// TwinCAT 3 PLC project LabExercise
// ProgramVersion: 3.1.4023.0
// libraries:
//   Tc2_NCI, * (Beckhoff Automation GmbH)
//   Tc2_Standard, * (Beckhoff Automation GmbH)
//   Tc2_System, * (Beckhoff Automation GmbH)
//   Tc3_Module, * (Beckhoff Automation GmbH)
//   VisuDialogs, * (System)
// project tree:
//   Comissioning/Function blocks/ FB_ModifyAutomaticControlSettings.TcPOU (not stored)
//   Comissioning/GVLs/ G_Commissioning.TcGVL (not stored)
//   Comissioning/Struct/ ST_AutomaticControlSettings.TcDUT (not stored), ST_ClosedLoopControlSettings.TcDUT (not stored), ST_MotionReferenceGeneratorSettings.TcDUT (not stored), ST_OpenLoopControlSettings.TcDUT (not stored)
//   ControlBox/Interfaces/ I_ControlBox.TcIO (not stored)
//   ControlBox/Function blocks/ FB_ControlBox.TcPOU, FB_RealControlBox.TcPOU (not stored), FB_VirtualControlBox.TcPOU (not stored)
//   CraneControl/Function blocks/Sub blocks/ FB_ActiveDamping.TcPOU (not stored), FB_Clock.TcPOU (not stored), FB_ClosedLoopControl.TcPOU (not stored), FB_Joystick.TcPOU (not stored), FB_MotionReferenceGenerator_limit.TcPOU (not stored), FB_OpenLoopControl.TcPOU (not stored), FB_ResetIntegralController.TcPOU (not stored), FB_Status.TcPOU (not stored)
//   CraneControl/Enums/ E_Mode.TcDUT (not stored), E_Status.TcDUT (not stored)
//   CraneControl/Function blocks/Main blocks/ FB_AutomaticControl.TcPOU (not stored), FB_ManualControl.TcPOU (not stored)
//   CraneControl/Functions/ F_BarToEng.TcPOU (not stored), F_LminToEng.TcPOU (not stored), F_RadToDeg.TcPOU (not stored)
//   CraneControl/GVLs/ G_Parameters.TcGVL (not stored), G_Work.TcGVL (not stored)
//   CraneControl/Struct/ ST_ActiveDamping.TcDUT (not stored), ST_Parameters.TcDUT (not stored)
//   / GlobalTextList.TcGTLO (not stored), PlcTask.TcTTO (not stored), Simulator.TcTTO (not stored), Visualization Manager.TcVMO (not stored)
//   HMI/ HMI.TcVIS (not stored)
//   HMI/Sub/ CommissioningHMI.TcVIS (not stored), VirtualControlBox.TcVIS (not stored)
//   Inputs/ FB_JoystickInputScaling.TcPOU (not stored), FB_PositionInputScaling.TcPOU (not stored), FB_PressureInputScaling.TcPOU (not stored), G_Inputs.TcGVL (not stored), G_Sensors.TcGVL (not stored)
//   Inputs/Struct/ ST_AnalogInput.TcDUT (not stored), ST_AnalogInputStatus.TcDUT (not stored)
//   Internship/ FB_ControlBlock.TcPOU, FB_SpeedProfile.TcPOU, F_PressureSensorInToBar.TcPOU (not stored), GVL_191759331.TcGVL, V2Q2u.TcPOU (not stored)
//   Outputs/ FB_ValveOutput.TcPOU (not stored), G_Outputs.TcGVL (not stored)
//   Outputs/Struct/ ST_pValveDeadBand.TcDUT (not stored), ST_ValveOutput.TcDUT (not stored)
//   ControlBox/GVLs/ G_VirtualControlBox.TcGVL (not stored)
//   Programs/ MAIN.TcPOU (not stored), P_ControlBlock.TcPOU, P_Commissioning.TcPOU (not stored), P_ControlBox.TcPOU (not stored), P_CraneControl.TcPOU (not stored), P_Inputs.TcPOU (not stored), P_OutputNonCompensated.TcPOU (not stored), P_Outputs.TcPOU (not stored), P_Simulator.TcPOU
//   Simulator/ FB_CraneSimulator.TcPOU (not stored), G_Simulator.TcGVL (not stored)
// real-time tasks:
//   TASK PlcTask: cycle T#1ms, priority 20, ADS port 350
//   TASK Simulator: cycle T#100us, priority 1, ADS port 351
// I/O:
//   DEVICE Device 5 (EtherCAT), AmsNetId 10.229.3.117.6.1
//     RIO (EK1100) [EK1100 EtherCAT Coupler (2A E-Bus)]
//       DI (EL1008) [EL1008 8Ch. Dig. Input 24V, 3ms]
//       DO (EL2008) [EL2008 8Ch. Dig. Output 24V, 0.5A]
//       AI1 (EL3068) [EL3068 8Ch. Ana. Input 0-10V]
//       AI2 (EL3068) [EL3068 8Ch. Ana. Input 0-10V]
//       AI3 (EL3174) [EL3174 4Ch. Ana. Input +/-10V Diff., +/-20mA SingleEnded, 16 Bit]
//       AO (EL4104) [EL4104 4Ch. Ana. Output 0-10V, 16bit]
//       End Cap (EL9011) [EL9011 End Terminal]
// variable links:
//   LabExercise/LabExercise Instance <-> Device 5 (EtherCAT)/RIO (EK1100)/AI1 (EL3068)
//     PlcTask Inputs/G_Inputs.stCylPos.nValue <-> AI Standard Channel 3/Value
//     PlcTask Inputs/G_Inputs.stCylPos.stStatus <-> AI Standard Channel 3/Status
//     PlcTask Inputs/G_Inputs.stJoyX.nValue <-> AI Standard Channel 1/Value
//     PlcTask Inputs/G_Inputs.stJoyX.stStatus <-> AI Standard Channel 1/Status
//     PlcTask Inputs/G_Inputs.stJoyY.nValue <-> AI Standard Channel 2/Value
//     PlcTask Inputs/G_Inputs.stJoyY.stStatus <-> AI Standard Channel 2/Status
//     PlcTask Inputs/G_Inputs.stSpoolPos.nValue <-> AI Standard Channel 4/Value
//     PlcTask Inputs/G_Inputs.stSpoolPos.stStatus <-> AI Standard Channel 4/Status
//   LabExercise/LabExercise Instance <-> Device 5 (EtherCAT)/RIO (EK1100)/AI2 (EL3068)
//     PlcTask Inputs/G_Inputs.stPressureCompensator.nValue <-> AI Standard Channel 3/Value
//     PlcTask Inputs/G_Inputs.stPressureCompensator.stStatus <-> AI Standard Channel 3/Status
//     PlcTask Inputs/G_Inputs.stPressureLhvSide.nValue <-> AI Standard Channel 5/Value
//     PlcTask Inputs/G_Inputs.stPressureLhvSide.stStatus <-> AI Standard Channel 5/Status
//     PlcTask Inputs/G_Inputs.stPressurePistonSide.nValue <-> AI Standard Channel 4/Value
//     PlcTask Inputs/G_Inputs.stPressurePistonSide.stStatus <-> AI Standard Channel 4/Status
//     PlcTask Inputs/G_Inputs.stPressureReturn.nValue <-> AI Standard Channel 2/Value
//     PlcTask Inputs/G_Inputs.stPressureReturn.stStatus <-> AI Standard Channel 2/Status
//     PlcTask Inputs/G_Inputs.stPressureRodSide.nValue <-> AI Standard Channel 6/Value
//     PlcTask Inputs/G_Inputs.stPressureRodSide.stStatus <-> AI Standard Channel 6/Status
//     PlcTask Inputs/G_Inputs.stPressureSupply.nValue <-> AI Standard Channel 1/Value
//     PlcTask Inputs/G_Inputs.stPressureSupply.stStatus <-> AI Standard Channel 1/Status
//   LabExercise/LabExercise Instance <-> Device 5 (EtherCAT)/RIO (EK1100)/AI3 (EL3174)
//     PlcTask Inputs/G_Inputs.stFlowReturnSide.nValue <-> AI Standard Channel 1/Value
//     PlcTask Inputs/G_Inputs.stFlowReturnSide.stStatus <-> AI Standard Channel 1/Status
//   LabExercise/LabExercise Instance <-> Device 5 (EtherCAT)/RIO (EK1100)/AO (EL4104)
//     PlcTask Outputs/G_Outputs.stValveOutput.nValveOutput <-> AO Output Channel 1/Analog output
//   LabExercise/LabExercise Instance <-> Device 5 (EtherCAT)/RIO (EK1100)/DI (EL1008)
//     PlcTask Inputs/G_Inputs.bAutoModeSelector <-> Channel 1/Input
//     PlcTask Inputs/G_Inputs.bManualModeSelector <-> Channel 2/Input
//     PlcTask Inputs/G_Inputs.bStartButton <-> Channel 3/Input
//     PlcTask Inputs/G_Inputs.bStopButton <-> Channel 4/Input
//   LabExercise/LabExercise Instance <-> Device 5 (EtherCAT)/RIO (EK1100)/DO (EL2008)
//     PlcTask Outputs/G_Outputs.bGreenLight <-> Channel 1/Output
//     PlcTask Outputs/G_Outputs.bRedLight <-> Channel 2/Output
//     PlcTask Outputs/G_Outputs.stValveOutput.bEnable <-> Channel 3/Output

// ---- Internship/GVL_191759331.TcGVL
VAR_GLOBAL CONSTANT
	SS_INITIALIZE: SINT := 0;
	SS_STEP: SINT := 1;
END_VAR

// ---- ControlBox/Function blocks/FB_ControlBox.TcPOU
FUNCTION_BLOCK FB_ControlBox
VAR_INPUT
	bRealControlBox : BOOL;
	eStatus : E_Status;
END_VAR
VAR_OUTPUT
	eMode : E_Mode;
END_VAR
VAR
	fbVirtualControlBox : FB_VirtualControlBox;
	fbRealControlBox : FB_RealControlBox;
	fbSelectedControlBox : I_ControlBox := fbVirtualControlBox;
END_VAR

IF bRealControlBox THEN
	fbSelectedControlBox := fbRealControlBox;
	//fbSelectedControlBox := fbVirtualControlBox;
ELSE
	fbSelectedControlBox := fbVirtualControlBox;
END_IF	
	
fbSelectedControlBox.ModeSelector(
	eMode => eMode
);

fbSelectedControlBox.PushButtons(
	eMode := eMode,
	eStatus := eStatus,
	bStart => G_Work.bStartButton,
	bStop => G_Work.bStopButton 	
);

fbSelectedControlBox.Lamps(
	eMode := eMode,
	eStatus := eStatus
);

fbSelectedControlBox.Joystick(
	eMode := eMode,
	eStatus := eStatus,
	fJoystickY => G_Work.fJoystickY
);

END_FUNCTION_BLOCK

// ---- Internship/FB_ControlBlock.TcPOU
FUNCTION_BLOCK FB_ControlBlock
VAR_INPUT
	ssMethodType: SINT;
	X_real: LREAL;
	Pa: LREAL;
	Pb: LREAL;
	Ps: LREAL;
	Clock: LREAL;
END_VAR
VAR_OUTPUT
	u: LREAL;
END_VAR
VAR
	rtb_y: LREAL := FB_SpeedProfile.fXdot;
	
	rtb_DiscreteTransferFcn: LREAL;
	rtb_TSamp: LREAL;
	rtb_fPosError: LREAL;
	fPosError: LREAL;
	DiscreteTransferFcn1: LREAL;
	temp1: LREAL;
	temp2: LREAL;
	c_DiscreteTimeIntegrator_DS: LREAL;
	d_DiscreteTimeIntegrator_DS: LREAL;
	DiscreteTransferFcn_states: LREAL;
	DiscreteTransferFcn1_states: LREAL;
	DiscreteTransferFcn2_states: LREAL;
	DiscreteTransferFcn3_states: LREAL;
	c_DiscreteTransferFcn_state: LREAL;
	UD_DSTATE: LREAL;
END_VAR



CASE ssMethodType OF
    SS_INITIALIZE: 
        (* SystemInitialize for Atomic SubSystem: '<Root>/CTRL' *)
        (* InitializeConditions for DiscreteTransferFcn: '<S1>/Discrete Transfer Fcn' *)
        DiscreteTransferFcn_states := 0.0;
        (* InitializeConditions for DiscreteTransferFcn: '<S1>/Discrete Transfer Fcn1' *)
        DiscreteTransferFcn1_states := 0.0;
        (* InitializeConditions for DiscreteTransferFcn: '<S1>/Discrete Transfer Fcn2' *)
        DiscreteTransferFcn2_states := 0.0;
        (* InitializeConditions for DiscreteTransferFcn: '<S1>/Discrete Transfer Fcn3' *)
        DiscreteTransferFcn3_states := 0.0;
        (* InitializeConditions for DiscreteIntegrator: '<S1>/Discrete-Time Integrator' *)
        c_DiscreteTimeIntegrator_DS := 0.0;
        (* InitializeConditions for DiscreteTransferFcn: '<S2>/Discrete Transfer Fcn' *)
        c_DiscreteTransferFcn_state := 0.0;
        (* InitializeConditions for DiscreteIntegrator: '<S2>/Discrete-Time Integrator' *)
        d_DiscreteTimeIntegrator_DS := 0.0;
        (* InitializeConditions for UnitDelay: '<S5>/UD'
         *
         * Block description for '<S5>/UD':
         *  
         *  Store in Global RAM *)
        UD_DSTATE := 0.0;
        (* End of SystemInitialize for SubSystem: '<Root>/CTRL' *)
    SS_STEP: 
        (* Outputs for Atomic SubSystem: '<Root>/CTRL' *)
        (* DiscreteTransferFcn: '<S1>/Discrete Transfer Fcn' *)
        rtb_DiscreteTransferFcn := 0.09516 * DiscreteTransferFcn_states;
        (* DiscreteTransferFcn: '<S1>/Discrete Transfer Fcn1' *)
        DiscreteTransferFcn1 := 0.003137 * DiscreteTransferFcn1_states;
        (* Sum: '<S1>/fPosError' incorporates:
         *  DiscreteIntegrator: '<S1>/Discrete-Time Integrator' *)
        fPosError := c_DiscreteTimeIntegrator_DS - X_real;
        (* SampleTimeMath: '<S5>/TSamp' incorporates:
         *  DiscreteTransferFcn: '<S2>/Discrete Transfer Fcn'
         *
         * About '<S5>/TSamp':
         *  y = u * K where K = 1 / ( w * Ts )
         *   *)
        rtb_TSamp := (0.0009995 * c_DiscreteTransferFcn_state) * 5.0;
        (* Sum: '<S2>/fPosError' incorporates:
         *  DiscreteIntegrator: '<S2>/Discrete-Time Integrator'
         *  Gain: '<S2>/Kp1'
         *  Sum: '<S5>/Diff'
         *  UnitDelay: '<S5>/UD'
         *
         * Block description for '<S5>/Diff':
         *  
         *  Add in CPU
         *
         * Block description for '<S5>/UD':
         *  
         *  Store in Global RAM *)
		 
		 
		 (* PID Output = Kp * Error + Ki * int(Error) + Kd * dError *)
        rtb_fPosError := ((2.0 * fPosError) + d_DiscreteTimeIntegrator_DS) + (rtb_TSamp - UD_DSTATE);

        

        (* MATLAB Function: '<S1>/V2Q2u' incorporates:
         *  DiscreteTransferFcn: '<S1>/Discrete Transfer Fcn2'
         *  DiscreteTransferFcn: '<S1>/Discrete Transfer Fcn3' *)
        (* MATLAB Function 'CTRL/V2Q2u': '<S3>:1' *)
        (* '<S3>:1:3' phi = 0.7130; *)
        (* '<S3>:1:4' A = 33.1/100^2; *)
        (* Area *)
        (* '<S3>:1:5' BW = 0; *)
        (* deadband *)
        (* '<S3>:1:6' SpoolTravel = 7; *)
        (* Maximum Spool Travel *)
        (* '<S3>:1:7' a = (SpoolTravel-BW)/25; *)
        (* Valve Slope Characteristic [mm/(L/min)] *)
        (* '<S3>:1:8' dP_0 = 7e5; *)
        (* Pressure drop with compansator *)
        (* '<S3>:1:10' if x_dot > 0 *)

        IF rtb_y > 0.0 THEN 
            (* '<S3>:1:11' Q = x_dot * A; *)
            (* Wanted Flow *)
            (* '<S3>:1:12' dP = (Ps-Pa)*1e5; *)
            (* '<S3>:1:13' dp_ref = abs(dP_0/dP); *)
            (* dp_ref = 1; *)
            (* '<S3>:1:15' Q_star = (Q * sqrt(dp_ref)) * 6e4; *)
            (* Referance Flow [L/min] *)
            (* '<S3>:1:16' u = (Q_star * a + BW)/SpoolTravel; *)
            temp2 := ABS(700000.0 / ((DiscreteTransferFcn1 - (0.003137 * DiscreteTransferFcn2_states)) * 100000.0));
            u := (((SQRT(temp2) * (rtb_y * 0.00331)) * 60000.0) * 0.28) / 7.0;
            (* Control Signal [-1, 1] *)
        ELSIF rtb_y < 0.0 THEN 
            (* '<S3>:1:18' elseif x_dot < 0 *)
            (* '<S3>:1:19' Q = x_dot * (A*phi); *)
            (* Wanted Flow *)
            (* '<S3>:1:20' dP = (Ps-Pb)*1e5; *)
            (* '<S3>:1:21' dp_ref = abs(dP_0/dP); *)
            (* dp_ref = 1; *)
            (* '<S3>:1:23' Q_star = (Q * sqrt(dp_ref)) * 6e4; *)
            (* Referance Flow [L/min] *)
            (* '<S3>:1:24' u = (Q_star * a - BW)/SpoolTravel; *)
            temp1 := ABS(700000.0 / ((DiscreteTransferFcn1 - (0.003137 * DiscreteTransferFcn3_states)) * 100000.0));
            u := (((SQRT(temp1) * (rtb_y * 0.00236003)) * 60000.0) * 0.28) / 7.0;
            (* Control Signal [-1, 1] *)
        ELSE 
            (* '<S3>:1:26' else *)
            (* '<S3>:1:27' u = 0; *)
            u := 0.0;
        END_IF;

        (* End of MATLAB Function: '<S1>/V2Q2u' *)
        

        (* Update for DiscreteTransferFcn: '<S1>/Discrete Transfer Fcn' *)
        DiscreteTransferFcn_states := u - (-0.9048 * DiscreteTransferFcn_states);
        (* Update for DiscreteTransferFcn: '<S1>/Discrete Transfer Fcn1' *)
        DiscreteTransferFcn1_states := Ps - (-0.9969 * DiscreteTransferFcn1_states);
        (* Update for DiscreteTransferFcn: '<S1>/Discrete Transfer Fcn2' *)
        DiscreteTransferFcn2_states := Pa - (-0.9969 * DiscreteTransferFcn2_states);
        (* Update for DiscreteTransferFcn: '<S1>/Discrete Transfer Fcn3' *)
        DiscreteTransferFcn3_states := Pb - (-0.9969 * DiscreteTransferFcn3_states);
        (* Update for DiscreteIntegrator: '<S1>/Discrete-Time Integrator' *)
        c_DiscreteTimeIntegrator_DS := (0.2 * rtb_y) + c_DiscreteTimeIntegrator_DS;
        (* Update for DiscreteTransferFcn: '<S2>/Discrete Transfer Fcn' *)
        c_DiscreteTransferFcn_state := fPosError - (-0.999 * c_DiscreteTransferFcn_state);
        (* Update for DiscreteIntegrator: '<S2>/Discrete-Time Integrator' *)
        d_DiscreteTimeIntegrator_DS := (0.2 * fPosError) + d_DiscreteTimeIntegrator_DS;
        (* Update for UnitDelay: '<S5>/UD'
         *
         * Block description for '<S5>/UD':
         *  
         *  Store in Global RAM *)
        UD_DSTATE := rtb_TSamp;
        (* Outport: '<Root>/u' incorporates:
         *  Sum: '<S1>/Sum' *)
        u := rtb_DiscreteTransferFcn + rtb_fPosError;
        (* End of Outputs for SubSystem: '<Root>/CTRL' *)
END_CASE;

END_FUNCTION_BLOCK

// ---- Internship/FB_SpeedProfile.TcPOU
FUNCTION_BLOCK FB_SpeedProfile
VAR_INPUT
	fClock : LREAL;
END_VAR
VAR_OUTPUT
	fXdot : LREAL;
END_VAR
VAR
END_VAR


fXdot := 0.0;


        IF fClock >= 1.0 THEN 

            IF fClock < 2.0 THEN 
                (* '<S4>:1:26' elseif t < t2 *)
                (* ramp up speed *)
                (* '<S4>:1:27' y = x_0 + v_0*(t-t1) + v_ref*(t-t1); *)
                fXdot := (fClock - 1.0) * 0.1;
            ELSIF fClock < 3.0 THEN 
                (* '<S4>:1:28' elseif t < t3 *)
                (* holding speed *)
                (* '<S4>:1:29' y = x_0 + v_ref*t_ramp; *)
                fXdot := 0.1;
            ELSIF fClock < 4.0 THEN 
                (* '<S4>:1:30' elseif t < t4 *)
                (* ramping down speed *)
                (* '<S4>:1:31' y = x_0 + v_ref*t_ramp - v_ref*(t-t3); *)
                fXdot := 0.1 - ((fClock - 3.0) * 0.1);
            ELSIF fClock >= 5.0 THEN 

                IF fClock < 6.0 THEN 
                    (* '<S4>:1:35' elseif t < t6 *)
                    (* ramping down speed *)
                    (* '<S4>:1:36' y = x_0 - v_0*(t-t5) - v_ref*(t-t5); *)
                    fXdot := 0.0 - ((fClock - 5.0) * 0.1);
                ELSIF fClock < 7.0 THEN 
                    (* '<S4>:1:37' elseif t < t7 *)
                    (* holdin speed *)
                    (* '<S4>:1:38' y = x_0 - v_ref*t_ramp; *)
                    fXdot := -0.1;
                ELSIF fClock < 8.0 THEN 
                    (* '<S4>:1:39' elseif t < t8 *)
                    (* ramping up speed *)
                    (* '<S4>:1:40' y = x_0 - v_ref*t_ramp + v_ref*(t-t7); *)
                    fXdot := ((fClock - 7.0) * 0.1) - 0.1;
                END_IF;

            END_IF;

        END_IF;

END_FUNCTION_BLOCK

// ---- Programs/P_ControlBlock.TcPOU
PROGRAM P_ControlBlock
VAR
	fbControlBlock : FB_ControlBlock;
END_VAR

fbControlBlock(
	ssMethodType := BOOL_TO_SINT(G_VirtualControlBox.bGreenLight),
	X_real:= G_Sensors.fPistonPosition,
	Pa:= G_Sensors.fPressurePistonSide, 
	Pb := G_Sensors.fPressureRodSide,
	Ps:= G_Sensors.fPressureSupply,
	Clock := 1,
	u	=> G_Work.fControlOutputNormalized
);

END_PROGRAM

// ---- Programs/P_Simulator.TcPOU
PROGRAM P_Simulator
VAR
	fbCraneSimulator : FB_CraneSimulator;
END_VAR

fbCraneSimulator(
	ssMethodType := BOOL_TO_SINT(G_Simulator.bSimulatorOn),	//
	uDCV := G_Work.fControlOutputNormalized,				//
	ppbar => G_Simulator.fPistonSidePressure,				// P_A
	prbar => G_Simulator.fRodSidePressure, 					// P_B
	xm => G_Simulator.fPistonPosition						// Position
);

END_PROGRAM
